// TIA Portal project "DawidKania_Delay" (V14)

(* hardware
DEVICE "S7-1200 station_1"  S7-1200 Station
   slot 0: "Rack_0"  S7-1200 Rack  Rack  V1.0
   slot 1: "PLC_1"  CPU 1214C DC/DC/DC  6ES7 214-1AG31-0XB0  V3.0
*)

// ===== PLC "PLC_1"  CPU 1214C DC/DC/DC =====

ORGANIZATION_BLOCK "Main"   // OB1, SCL, ProgramCycle
TITLE = "Main Program Sweep (Cycle)"
{ S7_Optimized_Access := 'TRUE' }
VERSION : 0.1
   VAR_TEMP
      "counter" : DInt;
   END_VAR
BEGIN


   #"counter" := DINT#100_000;

   WHILE #"counter" >= DINT#0 DO
       #"counter" := #"counter" - DINT#1;
   END_WHILE;
END_ORGANIZATION_BLOCK